NodeFactory.AddNodeAsPrototype('Vision/Container Statistics/F_VN_MedianElementElementwise/F_VN_MedianElementElementwise_DINT', node_F_VN_MedianElementElementwise_DINT);
NodeFactory.AddNodeAsPrototype('Vision/Container Statistics/F_VN_MedianElementElementwise/F_VN_MedianElementElementwise_INT', node_F_VN_MedianElementElementwise_INT);
NodeFactory.AddNodeAsPrototype('Vision/Container Statistics/F_VN_MedianElementElementwise/F_VN_MedianElementElementwise_LREAL', node_F_VN_MedianElementElementwise_LREAL);
NodeFactory.AddNodeAsPrototype('Vision/Container Statistics/F_VN_MedianElementElementwise/F_VN_MedianElementElementwise_REAL', node_F_VN_MedianElementElementwise_REAL);
NodeFactory.AddNodeAsPrototype('Vision/Container Statistics/F_VN_MedianElementElementwise/F_VN_MedianElementElementwise_SINT', node_F_VN_MedianElementElementwise_SINT);
NodeFactory.AddNodeAsPrototype('Vision/Container Statistics/F_VN_MedianElementElementwise/F_VN_MedianElementElementwise_TcVnPoint2_DINT', node_F_VN_MedianElementElementwise_TcVnPoint2_DINT);
NodeFactory.AddNodeAsPrototype('Vision/Container Statistics/F_VN_MedianElementElementwise/F_VN_MedianElementElementwise_TcVnPoint2_LREAL', node_F_VN_MedianElementElementwise_TcVnPoint2_LREAL);
NodeFactory.AddNodeAsPrototype('Vision/Container Statistics/F_VN_MedianElementElementwise/F_VN_MedianElementElementwise_TcVnPoint2_REAL', node_F_VN_MedianElementElementwise_TcVnPoint2_REAL);
NodeFactory.AddNodeAsPrototype('Vision/Container Statistics/F_VN_MedianElementElementwise/F_VN_MedianElementElementwise_TcVnPoint3_LREAL', node_F_VN_MedianElementElementwise_TcVnPoint3_LREAL);
NodeFactory.AddNodeAsPrototype('Vision/Container Statistics/F_VN_MedianElementElementwise/F_VN_MedianElementElementwise_TcVnPoint3_REAL', node_F_VN_MedianElementElementwise_TcVnPoint3_REAL);
NodeFactory.AddNodeAsPrototype('Vision/Container Statistics/F_VN_MedianElementElementwise/F_VN_MedianElementElementwise_TcVnVector2_DINT', node_F_VN_MedianElementElementwise_TcVnVector2_DINT);
NodeFactory.AddNodeAsPrototype('Vision/Container Statistics/F_VN_MedianElementElementwise/F_VN_MedianElementElementwise_TcVnVector2_INT', node_F_VN_MedianElementElementwise_TcVnVector2_INT);
NodeFactory.AddNodeAsPrototype('Vision/Container Statistics/F_VN_MedianElementElementwise/F_VN_MedianElementElementwise_TcVnVector2_REAL', node_F_VN_MedianElementElementwise_TcVnVector2_REAL);
NodeFactory.AddNodeAsPrototype('Vision/Container Statistics/F_VN_MedianElementElementwise/F_VN_MedianElementElementwise_TcVnVector2_SINT', node_F_VN_MedianElementElementwise_TcVnVector2_SINT);
NodeFactory.AddNodeAsPrototype('Vision/Container Statistics/F_VN_MedianElementElementwise/F_VN_MedianElementElementwise_TcVnVector2_UINT', node_F_VN_MedianElementElementwise_TcVnVector2_UINT);
NodeFactory.AddNodeAsPrototype('Vision/Container Statistics/F_VN_MedianElementElementwise/F_VN_MedianElementElementwise_TcVnVector2_USINT', node_F_VN_MedianElementElementwise_TcVnVector2_USINT);
NodeFactory.AddNodeAsPrototype('Vision/Container Statistics/F_VN_MedianElementElementwise/F_VN_MedianElementElementwise_TcVnVector3_INT', node_F_VN_MedianElementElementwise_TcVnVector3_INT);
NodeFactory.AddNodeAsPrototype('Vision/Container Statistics/F_VN_MedianElementElementwise/F_VN_MedianElementElementwise_TcVnVector3_REAL', node_F_VN_MedianElementElementwise_TcVnVector3_REAL);
NodeFactory.AddNodeAsPrototype('Vision/Container Statistics/F_VN_MedianElementElementwise/F_VN_MedianElementElementwise_TcVnVector3_SINT', node_F_VN_MedianElementElementwise_TcVnVector3_SINT);
NodeFactory.AddNodeAsPrototype('Vision/Container Statistics/F_VN_MedianElementElementwise/F_VN_MedianElementElementwise_TcVnVector3_UINT', node_F_VN_MedianElementElementwise_TcVnVector3_UINT);
NodeFactory.AddNodeAsPrototype('Vision/Container Statistics/F_VN_MedianElementElementwise/F_VN_MedianElementElementwise_TcVnVector3_USINT', node_F_VN_MedianElementElementwise_TcVnVector3_USINT);
NodeFactory.AddNodeAsPrototype('Vision/Container Statistics/F_VN_MedianElementElementwise/F_VN_MedianElementElementwise_TcVnVector4_DINT', node_F_VN_MedianElementElementwise_TcVnVector4_DINT);
NodeFactory.AddNodeAsPrototype('Vision/Container Statistics/F_VN_MedianElementElementwise/F_VN_MedianElementElementwise_TcVnVector4_INT', node_F_VN_MedianElementElementwise_TcVnVector4_INT);
NodeFactory.AddNodeAsPrototype('Vision/Container Statistics/F_VN_MedianElementElementwise/F_VN_MedianElementElementwise_TcVnVector4_LREAL', node_F_VN_MedianElementElementwise_TcVnVector4_LREAL);
NodeFactory.AddNodeAsPrototype('Vision/Container Statistics/F_VN_MedianElementElementwise/F_VN_MedianElementElementwise_TcVnVector4_SINT', node_F_VN_MedianElementElementwise_TcVnVector4_SINT);
NodeFactory.AddNodeAsPrototype('Vision/Container Statistics/F_VN_MedianElementElementwise/F_VN_MedianElementElementwise_TcVnVector4_UINT', node_F_VN_MedianElementElementwise_TcVnVector4_UINT);
NodeFactory.AddNodeAsPrototype('Vision/Container Statistics/F_VN_MedianElementElementwise/F_VN_MedianElementElementwise_TcVnVector4_USINT', node_F_VN_MedianElementElementwise_TcVnVector4_USINT);
NodeFactory.AddNodeAsPrototype('Vision/Container Statistics/F_VN_MedianElementElementwise/F_VN_MedianElementElementwise_UDINT', node_F_VN_MedianElementElementwise_UDINT);
NodeFactory.AddNodeAsPrototype('Vision/Container Statistics/F_VN_MedianElementElementwise/F_VN_MedianElementElementwise_UINT', node_F_VN_MedianElementElementwise_UINT);
NodeFactory.AddNodeAsPrototype('Vision/Container Statistics/F_VN_MedianElementElementwise/F_VN_MedianElementElementwise_ULINT', node_F_VN_MedianElementElementwise_ULINT);
NodeFactory.AddNodeAsPrototype('Vision/Container Statistics/F_VN_MedianElementElementwise/F_VN_MedianElementElementwise_USINT', node_F_VN_MedianElementElementwise_USINT);

NodeFactory.AddNodeAsPrototype('Vision/Container Statistics/F_VN_MinElementElementwise/F_VN_MinElementElementwise_DINT', node_F_VN_MinElementElementwise_DINT);
NodeFactory.AddNodeAsPrototype('Vision/Container Statistics/F_VN_MinElementElementwise/F_VN_MinElementElementwise_INT', node_F_VN_MinElementElementwise_INT);
NodeFactory.AddNodeAsPrototype('Vision/Container Statistics/F_VN_MinElementElementwise/F_VN_MinElementElementwise_LREAL', node_F_VN_MinElementElementwise_LREAL);
NodeFactory.AddNodeAsPrototype('Vision/Container Statistics/F_VN_MinElementElementwise/F_VN_MinElementElementwise_REAL', node_F_VN_MinElementElementwise_REAL);
NodeFactory.AddNodeAsPrototype('Vision/Container Statistics/F_VN_MinElementElementwise/F_VN_MinElementElementwise_SINT', node_F_VN_MinElementElementwise_SINT);
NodeFactory.AddNodeAsPrototype('Vision/Container Statistics/F_VN_MinElementElementwise/F_VN_MinElementElementwise_TcVnPoint2_DINT', node_F_VN_MinElementElementwise_TcVnPoint2_DINT);
NodeFactory.AddNodeAsPrototype('Vision/Container Statistics/F_VN_MinElementElementwise/F_VN_MinElementElementwise_TcVnPoint2_LREAL', node_F_VN_MinElementElementwise_TcVnPoint2_LREAL);
NodeFactory.AddNodeAsPrototype('Vision/Container Statistics/F_VN_MinElementElementwise/F_VN_MinElementElementwise_TcVnPoint2_REAL', node_F_VN_MinElementElementwise_TcVnPoint2_REAL);
NodeFactory.AddNodeAsPrototype('Vision/Container Statistics/F_VN_MinElementElementwise/F_VN_MinElementElementwise_TcVnPoint3_LREAL', node_F_VN_MinElementElementwise_TcVnPoint3_LREAL);
NodeFactory.AddNodeAsPrototype('Vision/Container Statistics/F_VN_MinElementElementwise/F_VN_MinElementElementwise_TcVnPoint3_REAL', node_F_VN_MinElementElementwise_TcVnPoint3_REAL);
NodeFactory.AddNodeAsPrototype('Vision/Container Statistics/F_VN_MinElementElementwise/F_VN_MinElementElementwise_TcVnVector2_DINT', node_F_VN_MinElementElementwise_TcVnVector2_DINT);
NodeFactory.AddNodeAsPrototype('Vision/Container Statistics/F_VN_MinElementElementwise/F_VN_MinElementElementwise_TcVnVector2_INT', node_F_VN_MinElementElementwise_TcVnVector2_INT);
NodeFactory.AddNodeAsPrototype('Vision/Container Statistics/F_VN_MinElementElementwise/F_VN_MinElementElementwise_TcVnVector2_REAL', node_F_VN_MinElementElementwise_TcVnVector2_REAL);
NodeFactory.AddNodeAsPrototype('Vision/Container Statistics/F_VN_MinElementElementwise/F_VN_MinElementElementwise_TcVnVector2_SINT', node_F_VN_MinElementElementwise_TcVnVector2_SINT);
NodeFactory.AddNodeAsPrototype('Vision/Container Statistics/F_VN_MinElementElementwise/F_VN_MinElementElementwise_TcVnVector2_UINT', node_F_VN_MinElementElementwise_TcVnVector2_UINT);
NodeFactory.AddNodeAsPrototype('Vision/Container Statistics/F_VN_MinElementElementwise/F_VN_MinElementElementwise_TcVnVector2_USINT', node_F_VN_MinElementElementwise_TcVnVector2_USINT);
NodeFactory.AddNodeAsPrototype('Vision/Container Statistics/F_VN_MinElementElementwise/F_VN_MinElementElementwise_TcVnVector3_INT', node_F_VN_MinElementElementwise_TcVnVector3_INT);
NodeFactory.AddNodeAsPrototype('Vision/Container Statistics/F_VN_MinElementElementwise/F_VN_MinElementElementwise_TcVnVector3_REAL', node_F_VN_MinElementElementwise_TcVnVector3_REAL);
NodeFactory.AddNodeAsPrototype('Vision/Container Statistics/F_VN_MinElementElementwise/F_VN_MinElementElementwise_TcVnVector3_SINT', node_F_VN_MinElementElementwise_TcVnVector3_SINT);
NodeFactory.AddNodeAsPrototype('Vision/Container Statistics/F_VN_MinElementElementwise/F_VN_MinElementElementwise_TcVnVector3_UINT', node_F_VN_MinElementElementwise_TcVnVector3_UINT);
NodeFactory.AddNodeAsPrototype('Vision/Container Statistics/F_VN_MinElementElementwise/F_VN_MinElementElementwise_TcVnVector3_USINT', node_F_VN_MinElementElementwise_TcVnVector3_USINT);
NodeFactory.AddNodeAsPrototype('Vision/Container Statistics/F_VN_MinElementElementwise/F_VN_MinElementElementwise_TcVnVector4_DINT', node_F_VN_MinElementElementwise_TcVnVector4_DINT);
NodeFactory.AddNodeAsPrototype('Vision/Container Statistics/F_VN_MinElementElementwise/F_VN_MinElementElementwise_TcVnVector4_INT', node_F_VN_MinElementElementwise_TcVnVector4_INT);
NodeFactory.AddNodeAsPrototype('Vision/Container Statistics/F_VN_MinElementElementwise/F_VN_MinElementElementwise_TcVnVector4_LREAL', node_F_VN_MinElementElementwise_TcVnVector4_LREAL);
NodeFactory.AddNodeAsPrototype('Vision/Container Statistics/F_VN_MinElementElementwise/F_VN_MinElementElementwise_TcVnVector4_SINT', node_F_VN_MinElementElementwise_TcVnVector4_SINT);
NodeFactory.AddNodeAsPrototype('Vision/Container Statistics/F_VN_MinElementElementwise/F_VN_MinElementElementwise_TcVnVector4_UINT', node_F_VN_MinElementElementwise_TcVnVector4_UINT);
NodeFactory.AddNodeAsPrototype('Vision/Container Statistics/F_VN_MinElementElementwise/F_VN_MinElementElementwise_TcVnVector4_USINT', node_F_VN_MinElementElementwise_TcVnVector4_USINT);
NodeFactory.AddNodeAsPrototype('Vision/Container Statistics/F_VN_MinElementElementwise/F_VN_MinElementElementwise_UDINT', node_F_VN_MinElementElementwise_UDINT);
NodeFactory.AddNodeAsPrototype('Vision/Container Statistics/F_VN_MinElementElementwise/F_VN_MinElementElementwise_UINT', node_F_VN_MinElementElementwise_UINT);
NodeFactory.AddNodeAsPrototype('Vision/Container Statistics/F_VN_MinElementElementwise/F_VN_MinElementElementwise_ULINT', node_F_VN_MinElementElementwise_ULINT);
NodeFactory.AddNodeAsPrototype('Vision/Container Statistics/F_VN_MinElementElementwise/F_VN_MinElementElementwise_USINT', node_F_VN_MinElementElementwise_USINT);
//F_VN_ContainerAverage
//F_VN_ContainerAverageElementwise2
//F_VN_ContainerAverageElementwise3
//F_VN_ContainerAverageElementwise4
//F_VN_ContainerAverageVariance
//F_VN_ContainerAverageVarianceElementwise2
//F_VN_ContainerAverageVarianceElementwise3
//F_VN_ContainerAverageVarianceElementwise4
//F_VN_MaxElement
//F_VN_MedianElement
//F_VN_MinElement

// Contour Analysis
//F_VN_ApproximatePolygon
//F_VN_CheckIfPointIsInsideContour
//F_VN_ContourArea
//F_VN_ContourCenterOfMass
//F_VN_ContourCircularity
//F_VN_ContourConvexity
//F_VN_ContourEccentricity
//F_VN_ContourElongation
//F_VN_ContourExtremePoint
//F_VN_ContourInertiaRatio
//F_VN_ContourMoments
//F_VN_ContourOrientation
//F_VN_ContourOrientationExp
//F_VN_ContourPerimeter
//F_VN_ContourRoundness
//F_VN_ConvexHullPoints
//F_VN_ConvexHullPointsExp
//F_VN_ConvexityDefects
//F_VN_CustomElementWiseContainerOperation_ITcVnContainer
//F_VN_CustomElementWiseContainerOperation_ITcVnForwardIterator
//F_VN_EnclosingCircle
//F_VN_EnclosingRectangle
//F_VN_EnclosingTriangle
//F_VN_FitEllipse
NodeFactory.AddNodeAsPrototype('Vision/Contour Analysis/F_VN_FitLine', node_F_VN_FitLine);
//F_VN_FitLineExp
//F_VN_FourierDescriptors
//F_VN_MatchContours
//F_VN_MatchContours1vsN
//F_VN_MatchContours1vsNExp
//F_VN_MatchContoursExp
//F_VN_UprightBoundingRectangle

// Control Functions
//F_VN_StartAbsWatchdog
//F_VN_StartAbsWatchdogExp
//F_VN_StartRelWatchdog
//F_VN_StartRelWatchdogExp
//F_VN_StopWatchdog
    
// Drawing
//F_VN_DrawArrow
//F_VN_DrawArrow_TcVnVector4_DINT
//F_VN_DrawArrowExp
//F_VN_DrawArrowExp_TcVnVector4_DINT
NodeFactory.AddNodeAsPrototype('Vision/Drawing/F_VN_DrawCircle', node_F_VN_DrawCircle);
//F_VN_DrawCircleExp
//F_VN_DrawCircles
//F_VN_DrawCirclesExp
//F_VN_DrawCircularArc
//F_VN_DrawCircularArcExp
//F_VN_DrawComponents
//F_VN_DrawComponentsExp
NodeFactory.AddNodeAsPrototype('Vision/Drawing/F_VN_DrawContours', node_F_VN_DrawContours);
//F_VN_DrawContoursExp
//F_VN_DrawEllipse
//F_VN_DrawEllipseExp
//F_VN_DrawKeypoints
//F_VN_DrawKeypointsExp
NodeFactory.AddNodeAsPrototype('Vision/Drawing/F_VN_DrawLine', node_F_VN_DrawLine);
//F_VN_DrawLine_TcVnVector4_DINT
NodeFactory.AddNodeAsPrototype('Vision/Drawing/F_VN_DrawLine_TcVnVector4_LREAL', node_F_VN_DrawLine_TcVnVector4_LREAL);
//F_VN_DrawLineExp
//F_VN_DrawLineExp_TcVnVector4_DINT
//F_VN_DrawLineExp_TcVnVector4_LREAL
//F_VN_DrawLines
//F_VN_DrawLinesExp
//F_VN_DrawMatches
//F_VN_DrawMatchesExp
//F_VN_DrawOrientation
//F_VN_DrawOrientationExp
//F_VN_DrawPoint
//F_VN_DrawPointExp
//F_VN_DrawPoints
//F_VN_DrawPointsExp
//F_VN_DrawPolygon
//F_VN_DrawPolygonExp
//F_VN_DrawRectangle
//F_VN_DrawRectangle_TcVnRectangle_DINT
//F_VN_DrawRectangle_TcVnRectangle_UDINT
//F_VN_DrawRotatedRectangle
//F_VN_DrawRotatedRectangleExp
//F_VN_FillCircle
//F_VN_FillContours
//F_VN_FillEllipse
//F_VN_FillPolygon
//F_VN_FillRectangle
//F_VN_FillRotatedRectangle
//F_VN_PlotIntensityProfile
//F_VN_PlotIntensityProfileExp
NodeFactory.AddNodeAsPrototype('Vision/Drawing/F_VN_PutLabel', node_F_VN_PutLabel);
//F_VN_PutLabelExp
NodeFactory.AddNodeAsPrototype('Vision/Drawing/F_VN_PutText', node_F_VN_PutText);
//F_VN_PutTextExp

// Fourier Analysis
//F_VN_CreateBandpassButterworthFilter
//F_VN_CreateBandpassGaussianFilter
//F_VN_CreateBandrejectButterworthFilter
//F_VN_CreateBandrejectGaussianFilter
//F_VN_CreateHighpassButterworthFilter
//F_VN_CreateHighpassGaussianFilter
//F_VN_CreateLowpassButterworthFilter
//F_VN_CreateLowpassGaussianFilter
//F_VN_Dft
//F_VN_InverseDft
//F_VN_OptimalDftSize
//F_VN_PadImageBorder
//F_VN_PadImageBorderExp

// Geometric and Coordinate Transformations
//F_VN_CalibrateCamera
//F_VN_CalibrateCameraExp
//F_VN_CalibrateCameraExp2
//F_VN_CalibrateCameraExp3
//F_VN_CalibrateCameraManually
//F_VN_CalibrateCameraManuallyExp
//F_VN_CalibrateCameraPlanar
//F_VN_CalibrateCameraPlanarExp
//F_VN_CalibrateLinescanCamera
//F_VN_CalibrateLinescanCameraExp
//F_VN_CompensateLensDistortion
//F_VN_CompensateLensDistortionExp1
//F_VN_CompensateLensDistortionExp2
//F_VN_CompensateLensDistortionForPoints
//F_VN_CompensateLensDistortionForPointsExp1
//F_VN_CompensateLensDistortionForPointsExp2
//F_VN_DetectPatternPoints
//F_VN_DetectPatternPointsExp
//F_VN_GenerateCalibrationPatternReferencePoints
//F_VN_ImagePointsWorldDistance
//F_VN_SolvePnP
//F_VN_SolvePnPExp
//F_VN_SortDetectedPatternPoints
//F_VN_TransformCoordinatesImageToWorld_Container
//F_VN_TransformCoordinatesImageToWorld_Point
//F_VN_TransformCoordinatesPlanar_Container
//F_VN_TransformCoordinatesPlanar_Point
//F_VN_TransformCoordinatesWorldToImage_Container
//F_VN_TransformCoordinatesWorldToImage_Point
//F_VN_AlignRotatedImageRegion
//F_VN_AlignRotatedImageRegionExp
//F_VN_ApplyRotationToAffineTransformation
//F_VN_ApplyRotationToAffineTransformationExp
//F_VN_ApplyScalingToAffineTransformation
//F_VN_ApplyScalingToAffineTransformationExp
//F_VN_ApplyTranslationToAffineTransformation
//F_VN_ApplyTranslationToAffineTransformationExp
//F_VN_ApplyYAxisInversionToAffineTransformation
//F_VN_ApplyYAxisInversionToAffineTransformationExp
//F_VN_ConvertCartesianToPolarAngleImage
//F_VN_ConvertCartesianToPolarAngleImageExp
//F_VN_ConvertCartesianToPolarAngles
//F_VN_ConvertCartesianToPolarAnglesExp
//F_VN_ConvertCartesianToPolarImages
//F_VN_ConvertCartesianToPolarImagesExp
//F_VN_ConvertCartesianToPolarMagnitudeImage
//F_VN_ConvertCartesianToPolarMagnitudes
//F_VN_ConvertCartesianToPolarPoints
//F_VN_ConvertCartesianToPolarPointsExp
//F_VN_ConvertPolarToCartesianImages
//F_VN_ConvertPolarToCartesianImagesExp
//F_VN_ConvertPolarToCartesianPoints
//F_VN_ConvertPolarToCartesianPointsExp
//F_VN_DecomposeAffineTransformation
//F_VN_DecomposeAffineTransformationExp
//F_VN_DecomposeHomography
//F_VN_DecomposeHomographyExp
NodeFactory.AddNodeAsPrototype('Vision/Geometric and Coordinate Transformations/F_VN_FlipImage', node_F_VN_FlipImage);
//F_VN_GenerateAffineTransformationUnitMatrix2D
//F_VN_GetAffineTransformation
//F_VN_GetAffineTransformation2D
//F_VN_GetAffineTransformation2DExp
//F_VN_GetPerspectiveTransformation
//F_VN_Homography
//F_VN_HomographyExp
//F_VN_InvertAffineTransformation
//F_VN_PerspectiveTransformation
NodeFactory.AddNodeAsPrototype('Vision/Geometric and Coordinate Transformations/F_VN_PyramidDown', node_F_VN_PyramidDown);
NodeFactory.AddNodeAsPrototype('Vision/Geometric and Coordinate Transformations/F_VN_PyramidUp', node_F_VN_PyramidUp);
//F_VN_RemapImageToLogPolarSpace
//F_VN_RemapImageToLogPolarSpaceExp
//F_VN_RemapImageToLogPolarSpaceExp2
//F_VN_RemapImageToPolarSpace
//F_VN_RemapImageToPolarSpaceExp
//F_VN_RemapImageToPolarSpaceExp2
//F_VN_ResizeImage
//F_VN_ResizeImageExp
//F_VN_RotateImage
//F_VN_RotateImageExp
//F_VN_RotateImageExp2
//F_VN_WarpAffine
//F_VN_WarpAffine_Container
//F_VN_WarpAffine_Point
//F_VN_WarpAffine_Rectangle
//F_VN_WarpAffineExp
//F_VN_WarpPerspective
//F_VN_WarpPerspective_Container
//F_VN_WarpPerspective_Point
//F_VN_WarpPerspective_Rectangle
//F_VN_WarpPerspectiveExp

// Image Analysis
//F_VN_AdjustActiveContour
NodeFactory.AddNodeAsPrototype('Vision/Image Analysis/Object Detection/F_VN_DetectBlobs', node_F_VN_DetectBlobs);
//F_VN_DetectBlobsExp
//F_VN_FindContourHierarchyExp
//F_VN_FindContours
//F_VN_FindContoursExp
//F_VN_HoughCircles
//F_VN_HoughCirclesExp
//F_VN_HoughLines
//F_VN_HoughLinesExp
//F_VN_HoughLinesP
//F_VN_HoughLinesPExp
//F_VN_MatchImageHuMoments
//F_VN_MatchTemplate
//F_VN_MatchTemplateAndEvaluate
//F_VN_MatchTemplateAndEvaluateExp
//F_VN_MatchTemplateExp
//F_VN_CannyEdgeDetection
//F_VN_CannyEdgeDetectionExp
//F_VN_ConnectedComponents
//F_VN_ConnectedComponentsExp
//F_VN_ConnectedComponentsWithStats
//F_VN_ConnectedComponentsWithStatsExp
//F_VN_CountNonZeroPixels
NodeFactory.AddNodeAsPrototype('Vision/Image Analysis/F_VN_CountNonZeroPixels', node_F_VN_CountNonZeroPixels);
//F_VN_DistanceTransformation
//F_VN_DistanceTransformationExp
//F_VN_GetConnectedComponent
//F_VN_GetConnectedComponentExp
//F_VN_ImageAverage
//F_VN_ImageAverageExp
//F_VN_ImageAverageStdDev
//F_VN_ImageAverageStdDevExp
//F_VN_ImageCenterOfMass
//F_VN_ImageCenterOfMassExp
//F_VN_ImageMedian
//F_VN_ImageMedianExp
//F_VN_ImageMoments
//F_VN_MaxPixelValue
//F_VN_MaxPixelValueExp
//F_VN_MinPixelValue
//F_VN_MinPixelValueExp
//F_VN_RegionOrientation
//F_VN_RegionOrientationExp

// Image Color and Contrast Processing
NodeFactory.AddNodeAsPrototype('Vision/Image Color and Contrast Processing/F_VN_ApplyColorMap', node_F_VN_ApplyColorMap);
//F_VN_ApplyLut
//F_VN_Clahe
//F_VN_ClaheExp
NodeFactory.AddNodeAsPrototype('Vision/Image Color and Contrast Processing/F_VN_ConvertColorSpace', node_F_VN_ConvertColorSpace);
NodeFactory.AddNodeAsPrototype('Vision/Image Color and Contrast Processing/F_VN_GenerateColorMap', node_F_VN_GenerateColorMap);
//F_VN_GenerateCustomColorMap
//F_VN_Histogram
//F_VN_HistogramEqualization
//F_VN_HistogramEqualizationExp
//F_VN_HistogramExp
NodeFactory.AddNodeAsPrototype('Vision/Image Color and Contrast Processing/F_VN_InvertImageColor', node_F_VN_InvertImageColor);
//F_VN_InvertImageColorExp
NodeFactory.AddNodeAsPrototype('Vision/Image Color and Contrast Processing/F_VN_NormalizeImage', node_F_VN_NormalizeImage);
//F_VN_NormalizeImageExp
//F_VN_NormalizeImageForDisplay
//F_VN_ReferenceColorSimilarity_ITcVnColorModel
//F_VN_ReferenceColorSimilarity_ITcVnMlModel
//F_VN_ReferenceColorSimilarity_TcVnVector3_LREAL
//F_VN_ReferenceColorSimilarityExp_ITcVnColorModel
//F_VN_ReferenceColorSimilarityExp_ITcVnMlModel
//F_VN_ReferenceColorSimilarityExp_TcVnVector3_LREAL
//F_VN_TrainImageColor
//F_VN_TrainImageColor_ITcVnMlModel
//F_VN_TrainImageColorExp
//F_VN_TrainImageColorExp_ITcVnMlModel
//F_VN_TrainImageColorExp2
//F_VN_TrainImageColorExp2_ITcVnMlModel
//F_VN_WhiteBalance

// Image Filtering
//F_VN_BilateralFilter
//F_VN_BilateralFilterExp
NodeFactory.AddNodeAsPrototype('Vision/Image Filtering/F_VN_BoxFilter', node_F_VN_BoxFilter);
//F_VN_BoxFilterExp
NodeFactory.AddNodeAsPrototype('Vision/Image Filtering/F_VN_BrightBorderObjects', node_F_VN_BrightBorderObjects);
//F_VN_CreateStructuringElement
//F_VN_CustomFilter
//F_VN_CustomFilterExp
NodeFactory.AddNodeAsPrototype('Vision/Image Filtering/F_VN_DarkBorderObjects', node_F_VN_DarkBorderObjects);
NodeFactory.AddNodeAsPrototype('Vision/Image Filtering/F_VN_FillHoles', node_F_VN_FillHoles);
NodeFactory.AddNodeAsPrototype('Vision/Image Filtering/F_VN_GaussianFilter', node_F_VN_GaussianFilter);
//F_VN_GaussianFilterExp
NodeFactory.AddNodeAsPrototype('Vision/Image Filtering/F_VN_LaplacianFilter', node_F_VN_LaplacianFilter);
//F_VN_LaplacianFilterExp
NodeFactory.AddNodeAsPrototype('Vision/Image Filtering/F_VN_LocalMaxima', node_F_VN_LocalMaxima);
NodeFactory.AddNodeAsPrototype('Vision/Image Filtering/F_VN_LocalMinima', node_F_VN_LocalMinima);
//F_VN_MedianFilter
//F_VN_MorphologicalOperator
//F_VN_RemoveLocalMaxima
//F_VN_RemoveLocalMinima
//F_VN_ScharrFilter
//F_VN_ScharrFilterExp
//F_VN_SeparableCustomFilter
//F_VN_SeparableCustomFilterExp
//F_VN_SobelFilter
//F_VN_SobelFilterExp
//F_VN_VarianceFilter
//F_VN_VarianceFilterExp
    
// Image Segmentation
//F_VN_AdaptiveThreshold
//F_VN_AdaptiveThresholdExp
//F_VN_CheckColorRange
//F_VN_DoubleThreshold
NodeFactory.AddNodeAsPrototype('Vision/Image Segmentation/F_VN_Threshold', node_F_VN_Threshold);
//F_VN_WatershedSegmentationExp

// Keypoint Features
//F_VN_FilterGoodMatches
//F_VN_FindReferenceKeyPointsInImage
//F_VN_FindReferenceKeyPointsInImageAKAZE
//F_VN_FindReferenceKeyPointsInImageAKAZEExp
//F_VN_FindReferenceKeyPointsInImageBRISK
//F_VN_FindReferenceKeyPointsInImageBRISKExp
//F_VN_FindReferenceKeyPointsInImageExp
//F_VN_FindReferenceKeyPointsInImageORB
//F_VN_FindReferenceKeyPointsInImageORBExp
//F_VN_GetMatchCoordinates
NodeFactory.AddNodeAsPrototype('Vision/Keypoint Features/F_VN_KeyPointsAGAST', node_F_VN_KeyPointsAGAST);
//F_VN_KeyPointsAGASTExp
//F_VN_KeyPointsAndDescriptorsAKAZE
//F_VN_KeyPointsAndDescriptorsAKAZEExp
//F_VN_KeyPointsAndDescriptorsBRISK
//F_VN_KeyPointsAndDescriptorsBRISKExp
//F_VN_KeyPointsAndDescriptorsKAZE
//F_VN_KeyPointsAndDescriptorsKAZEExp
//F_VN_KeyPointsAndDescriptorsORB
//F_VN_KeyPointsAndDescriptorsORBExp
NodeFactory.AddNodeAsPrototype('Vision/Keypoint Features/F_VN_KeyPointsFAST', node_F_VN_KeyPointsFAST);
//F_VN_KeyPointsFASTExp
NodeFactory.AddNodeAsPrototype('Vision/Keypoint Features/F_VN_KeyPointsGFTT', node_F_VN_KeyPointsGFTT);
//F_VN_KeyPointsGFTTExp
NodeFactory.AddNodeAsPrototype('Vision/Keypoint Features/F_VN_KeyPointsMSER', node_F_VN_KeyPointsMSER);
//F_VN_KeyPointsMSERExp
NodeFactory.AddNodeAsPrototype('Vision/Keypoint Features/F_VN_KeyPointsSB', node_F_VN_KeyPointsSB);
//F_VN_KeyPointsSBExp
//F_VN_MatchDescriptorsBF
//F_VN_MatchDescriptorsBFExp
//F_VN_MatchDescriptorsFlannLsh
//F_VN_MatchDescriptorsFlannLshExp
//F_VN_MatchDescriptorsKnnBF
//F_VN_MatchDescriptorsKnnBFExp
//F_VN_MatchDescriptorsKnnFlannLsh
//F_VN_MatchDescriptorsKnnFlannLshExp
//F_VN_RegionsMSER
//F_VN_RegionsMSERExp

// Machine Learning
//F_VN_CreateBoostClassifier
//F_VN_CreateBoostClassifierExp
//F_VN_CreateBoostClassifierExp2
//F_VN_CreateKmppModel
//F_VN_CreateKmppModelExp
//F_VN_CreateKnnModel
//F_VN_CreateLbgModel
//F_VN_CreateLbgModelExp
//F_VN_CreateLdaTransform
//F_VN_CreateLdaTransformViaComponentNum
//F_VN_CreateNbcModel
//F_VN_CreatePcaTransform
//F_VN_CreatePcaTransformViaComponentNum
//F_VN_CreatePcaTransformViaVariance
//F_VN_CreateRTreesModel
//F_VN_CreateRTreesModelExp
//F_VN_CreateRTreesModelExp2
//F_VN_CreateStaModel
//F_VN_CreateStaModelExp
//F_VN_CreateStaModelExp2
//F_VN_CreateSvmModel
//F_VN_CreateSvmModelExp
//F_VN_CreateSvmModelExp2
//F_VN_CreateSvmSgdClassifier
//F_VN_CreateSvmSgdClassifierExp
//F_VN_FeatureScaling
//F_VN_FeatureScalingExp
//F_VN_FeatureTransform
//F_VN_GetBatchClusters
//F_VN_GetBatchClustersExp
//F_VN_GetBatchNovelties
//F_VN_GetClusterCenter
//F_VN_GetClusterNum
//F_VN_GetFeatureScales
//F_VN_GetSampleCluster
//F_VN_GetSampleClusterExp
//F_VN_GetSampleNovelty
//F_VN_InverseFeatureScaling
//F_VN_InverseFeatureScaling_REAL
//F_VN_InverseFeatureScalingExp
//F_VN_InverseFeatureScalingExp_REAL
//F_VN_InverseFeatureTransform
//F_VN_PredictBatch
//F_VN_PredictBatchExp
//F_VN_PredictSampleClass
//F_VN_PredictSampleClassExp
//F_VN_PredictSampleScalar
//F_VN_PredictSampleScalarExp
//F_VN_PredictSampleVector
//F_VN_PredictSampleVectorExp
//F_VN_TrainBatch
//F_VN_TrainBatchClusters
//F_VN_TrainSample
//F_VN_TrainSampleClass
//F_VN_TrainSampleCluster
//F_VN_TrainSampleScalar
//F_VN_TrainSampleVector

// Measurement
//F_VN_AdjustSearchWindowOrientationToLinearEdge
//F_VN_ClosestPointsBF
//F_VN_LocateCircularArc
//F_VN_LocateCircularArcExp
NodeFactory.AddNodeAsPrototype('Vision/Measurement/F_VN_LocateEdge', node_F_VN_LocateEdge);
NodeFactory.AddNodeAsPrototype('Vision/Measurement/F_VN_LocateEdgeExp', node_F_VN_LocateEdgeExp);
NodeFactory.AddNodeAsPrototype('Vision/Measurement/F_VN_LocateEdges', node_F_VN_LocateEdges);
NodeFactory.AddNodeAsPrototype('Vision/Measurement/F_VN_LocateEdgesExp', node_F_VN_LocateEdgesExp);
NodeFactory.AddNodeAsPrototype('Vision/Measurement/F_VN_LocateEllipse', node_F_VN_LocateEllipse);
//F_VN_LocateEllipseExp
//F_VN_MeasureAngleBetweenEdges
//F_VN_MeasureAngleBetweenEdgesExp
//F_VN_MeasureEdgeDistance
//F_VN_MeasureEdgeDistanceExp
//F_VN_MeasureMinEdgeDistance
//F_VN_MeasureMinEdgeDistanceExp

// Miscellaneous
//F_VN_CheckFunctionInitialization
//F_VN_ClipLineToBoundary
//F_VN_ClipLineToBoundary_ITcVnImage
//F_VN_ClipLineToBoundary_TcVnRectangle_DINT
//F_VN_ConvertITcUnknownToITcVnBitmapExport
//F_VN_ConvertITcUnknownToITcVnContainer
//F_VN_ConvertITcUnknownToITcVnImage
//F_VN_ConvertITcUnknownToITcVnMlModel
//F_VN_DeinitializeFunction
//F_VN_GetTimestamp
//F_VN_HuMomentInvariants
//F_VN_InitMatrixStruct
//F_VN_InvertMatrix3x3
//F_VN_LineIntersectionPoint
//F_VN_LineIntersectionPointAndAngle
//F_VN_MultiplyMatrices
//F_VN_RotatedRectangleCorners
//F_VN_RotatedRectangleIntersection
//F_VN_SetRngSeed
//F_VN_UpdateTimestamp

// OCR
//F_VN_OCR
//F_VN_OCRExp

// Texture Analysis
//F_VN_Granulometry
//F_VN_HaralickFeatures
END_METHOD

END_FUNCTION_BLOCK

// ---- VisionPack.TcPOU
{attribute 'linkalways'} 
{attribute 'no_explicit_call' := 'This FB is a CLASS and must be accessed using methods or properties'}
{attribute 'enable_dynamic_creation'}
FUNCTION_BLOCK VisionPack IMPLEMENTS I_GraphPack
VAR
	visionDatatypePack : VisionDatatypePack;
	visionNodePack : VisionNodePack;
END_VAR

METHOD RegisterWithDatatypes
VAR_INPUT
	Datatypes : I_Datatypes;
END_VAR
visionDatatypePack.RegisterWithDatatypes(Datatypes);
END_METHOD

METHOD PUBLIC RegisterWithNodeFactory
VAR_INPUT
	NodeFactory : I_NodeFactory;
END_VAR
visionNodePack.RegisterWithNodeFactory(NodeFactory);
END_METHOD

END_FUNCTION_BLOCK
